// TIA Portal V19 export
TYPE "typePressureGuageRs485AnalogProcessValues"
TITLE = LBC_typeAnalogProcessValues
// Module related monitoring information
// stored: Access Published
   STRUCT
      enable { ExternalWritable := 'False'} : Bool;   // Manual mode parameters for axis control interface
      referenceDesignator { ExternalWritable := 'False'} : WString[154];   // Reference Designator for the module incl. its parent
      simulation { ExternalWritable := 'False'} : Bool;   // Manual mode parameters for axis control interface
      processValue { ExternalWritable := 'False'} : LReal;   // Scaled process value
      analogValue { ExternalWritable := 'False'} : Int;   // Analog value for/from hardware periphery
      limitHigh2 { ExternalWritable := 'False'} : Bool;   // Manual mode parameters for axis control interface
      limitHigh1 { ExternalWritable := 'False'} : Bool;   // Manual mode parameters for axis control interface
      limitLow1 { ExternalWritable := 'False'} : Bool;   // Manual mode parameters for axis control interface
      limitLow2 { ExternalWritable := 'False'} : Bool;   // Manual mode parameters for axis control interface
      maxValueReached { ExternalWritable := 'False'} : Bool;   // Manual mode parameters for axis control interface
      minValueReached { ExternalWritable := 'False'} : Bool;   // Manual mode parameters for axis control interface
      error { ExternalWritable := 'False'} : Bool;   // Manual mode parameters for axis control interface
      status { ExternalWritable := 'False'} : Word;   // 16#0000-16#7FFF: Status of the FB 16#8000-16#FFFF: Error identification
   END_STRUCT;
END_TYPE
